{attribute 'qualified_only'}
VAR_GLOBAL
	MainJibPistForce : LREAL;
END_VAR

(* stored: Version 1.1.0.1, ProductVersion 3.1.4024.9
   GVL ToUnreal: Id {65dfc488-1564-4dc7-bf95-af1a545cd988} *)
